INTERFACE I_Brake

PROPERTY BrakeOpen : BOOL
GET
END_GET
END_PROPERTY

METHOD CloseBrake : BOOL
VAR_INPUT
END_VAR
END_METHOD

METHOD OpenBrake : BOOL
VAR_INPUT
END_VAR
END_METHOD

END_INTERFACE

(* stored: Version 1.1.0.1, ProductVersion 3.1.4026.11
   Itf I_Brake: Id {1ea40e6b-7b15-4224-8327-2c0169da68d6}
   Property BrakeOpen: Id {e9b670f4-c3dd-4a6c-b452-216be4638562}
   Get Get: Id {ead55009-18f9-4895-a1e0-d4cbb81f3778}
   Method CloseBrake: Id {0fa19818-81a5-4563-a75a-2ae1429c657d}
   Method OpenBrake: Id {61c25982-5a7c-403f-8b9e-e60c42fa6606} *)
